(* IEC 61131-3 sources: Hal/Libraries/sprintf, 3 files *)

(* ---- sprintf.typ ---- *)
(********************************************************************
 * COPYRIGHT -- B&R
 ********************************************************************
 * Library: sprintf
 * File: sprintf.typ
 * Author: buchananw
 * Created: April 15, 2009
 ********************************************************************
 * Data types of library sprintf
 ********************************************************************)

TYPE

END_TYPE

(* ---- sprintf.fun ---- *)
(********************************************************************
 * COPYRIGHT -- B&R
 ********************************************************************
 * Library: sprintf
 * File: sprintf.fun
 * Author: buchananw
 * Created: April 15, 2009
 ********************************************************************
 * Functions and function blocks of library sprintf
 ********************************************************************)

FUNCTION sprintf2 : INT
END_FUNCTION

FUNCTION snprintf2 : INT
END_FUNCTION

(* ---- sprintf.var ---- *)
(********************************************************************
 * COPYRIGHT -- B&R
 ********************************************************************
 * Library: sprintf
 * File: sprintf.var
 * Author: buchananw
 * Created: April 15, 2009
 ********************************************************************
 * Constants of library sprintf
 ********************************************************************)

VAR CONSTANT

END_VAR
